// TIA Portal project "User_Management" (V17)

(* hardware
DEVICE "HMI_1"  KTP700 Basic PN
   slot 0: "HMI_1"  KTP700 Basic PN  6AV2 123-2GB03-0AX0  17.0.0.0
   slot 1: "HMI_RT_1"  KTP700 Basic PN  6AV2 123-2GB03-0AX0  17.0.0.0
   slot 5: "HMI_1.IE_CP_1"  PROFINET Interface  17.0.0.0
      slot 1: "PROFINET Interface_1"  PROFINET Interface
         slot 1: "Port_1"  Port
DEVICE "S7-1200 station_1"  S7-1200 Station
   slot 0: "Rack_0"  S7-1200 Rack  Rack  V1.0
   slot 1: "PLC_1"  CPU 1215C DC/DC/DC  6ES7 215-1AG40-0XB0  V4.5
*)

// ===== PLC "PLC_1"  CPU 1215C DC/DC/DC =====

VAR_GLOBAL   // PLC tag table "Default tag table"
   "HMI Start Stop Button" AT %M10.0 : Bool;
   "Mixer" AT %Q0.0 : Bool;
END_VAR

ORGANIZATION_BLOCK "Main"   // OB1, LAD, ProgramCycle
TITLE = "Main Program Sweep (Cycle)"
{ S7_Optimized_Access := 'TRUE' }
VERSION : 0.1
   VAR_INPUT
      Initial_Call : Bool;   // Initial call of this OB
      Remanence : Bool;   // =True, if remanent data are available
   END_VAR
BEGIN

REGION Network 1
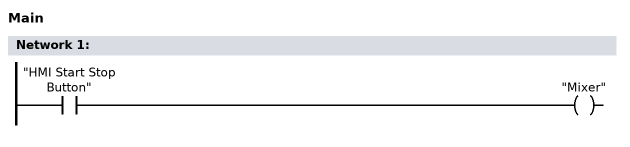
   RUNG wire#powerrail
      Contact( "HMI Start Stop Button" )
      Coil( "Mixer" )
   END_RUNG
   // the same network as SCL:
   "Mixer" := "HMI Start Stop Button";
END_REGION
END_ORGANIZATION_BLOCK

(* ===== HMI "HMI_RT_1" =====
system functions are stored by id; their names below are inferred from use
connection "HMI_Connection_1": ETHERNET, SMART_S7_1200_OMS

HMI tags "Default tag table"
   "Mixer" : Bool = PLC Mixer AT %Q0.0, 1 s
   "HMI Start Stop Button" : Bool = PLC "HMI Start Stop Button" AT %M10.0, 1 s

graphic list "Graphic_list_1": 0 'Graphic_1'; 1 'Graphic_2'

screen "User Screen" 800x480, template "Template_1"
   TextField "Text field_1" at 260,9 size 265x32; Text 'USER ACCESS SCREEN'
   Button "Button_1" at 174,144 size 116x44; TextOff 'LOG ON'
      on Press: function_a2a04561()
   Button "Button_3" at 471,144 size 116x44; TextOff 'LOG OFF'
      on Press: function_f23ef4c9()
   Button "Button_2" at 718,420 size 60x50; TextOff 'Text'; PictureOff "Right_Arrow"; Authorization "Monitor"
      on Press: ActivateScreen("Control Screen", 0)

screen "Control Screen" 800x480
   TextField "Text field_1" at 282,9 size 218x32; Text 'CONTROL SCREEN'
   Button "Button_1" at 191,155 size 142x63; TextOff 'START/STOP'; Authorization "Operate"
      on Press: InvertBit("HMI Start Stop Button")
   GraphicIOField "Graphic I/O field_1" at 529,127 size 91x167; PictureList "Graphic_list_1"
      ProcessValue <- "Mixer"
   Button "Button_2" at 20,420 size 60x50; TextOff 'Text'; PictureOff "Left_Arrow"; Authorization "Monitor"
      on Press: ActivateScreen("User Screen", 0)
   Button "Button_3" at 718,420 size 60x50; TextOff 'Text'; PictureOff "Right_Arrow"; Authorization "User administration"
      on Press: ActivateScreen("User Management Screen", 0)

screen "User Management Screen" 800x480
   UserView "User view_1" at 14,118 size 758x196
   TextField "Text field_1" at 242,9 size 344x32; Text 'USER MANAGEMENT SCREEN'
   Button "Button_2" at 20,420 size 60x50; TextOff 'Text'; PictureOff "Left_Arrow"; Authorization "User administration"
      on Press: ActivateScreen("Control Screen", 0)
*)